# EPICS substitutions: examples/test/el6022/ecmcEL6022_bytes.substitutions
file "ecmcEcSlave.template"
{
  pattern {}
          {}
}

file "ecmcEL6022-chX_bytes.template"
{
  pattern {CH_ID, PLC_ID, NELM }
          {01,    0,      22   }
          {02,    1,      22   }
}
